{attribute 'qualified_only'}
{attribute 'strict'}
{attribute 'to_string'}
TYPE ST150_Uss_e :
(
    RESET := 0, // Reset

    INIT := 100, // Initialisieren 
    Init_ResetUss_maintaining_down,

    READY := 999,  // READY to Start, Init Done 
    START := 1000, // Start Zyklisch
    MOVER_FREE_OP, // Ab here, operation without mover can be done

    waitOnMover,     // wait until the mover is there
    MOVER_NEEDED_OP, // Since here, a mover in position is needed to perform the action

    check_cap_present,     // See if the sensor sees the cap
    mover_maintening_up,   // Kraftbstützung goes up
    uss_start,             // start signal is given
    uss_working,           // we wait until the uss is finished
    mover_maintening_down, // Kraftbstützung goes down

    SYNC_MOVER_LEAVE, // MoverMan need to take the mover
    DONE := 8000,     // Ablauf beendet 
    ERROR := 9000,    // Fehler 
    _max
);
END_TYPE

(* stored: Version 1.1.0.1, ProductVersion 3.1.4024.6
   EnumerationTextList ST150_Uss_e: Id {70f6ed33-469a-49d2-9229-880d3ad30ccd} *)
